(* Schneider Machine Expert - Basic project resolucao, file version 2.7.0.0 *)
(* ProjectInformations: Name=Novo projeto *)

HARDWARE
  Cpu 0: TM221CE24R
  EthernetConfiguration: NetworkName=M221, IpAllocationMode=FixedAddress, IpAddress=0.0.0.0, SubnetMask=0.0.0.0
  SerialLineConfiguration: Baud=Baud19200, Parity=ParityEven, DataBits=DataBits8, StopBits=StopBits1, PhysicalMedium=PhysicalMediumRs485, TransmissionMode=TransmissionModeModbusRtu, SlaveId=1, Addressing=SlaveAddressing
  MastTask: UsePeriodScanMode=false, PeriodScan=100
  FastTask: Period=255
  CpuBehavior: StartingMode=StartAsPreviousState, AutoSaveRamOnEeprom=true, WatchdogPeriod=250

SYMBOLS  (address, symbol, comment, settings)
  %M0       SIG_IN_BOT_G
  %M10      SIG_OUT_CON_A_LIGA
  %M11      SIG_OUT_CON_A_DESL
  %M12      SIG_OUT_MOT_E_LIGA
  %M13      SIG_OUT_MOT_E_DESL
  %TM0      T_CON_A_LIGA  [Preset=5, Base=OneHundredMilliSeconds]
  %TM1        [Preset=5, Base=OneHundredMilliSeconds]
  %I0.0     IN_BOT_G
  %Q0.1     OUT_CON_A
  %Q0.2     OUT_MOT_E

POU Entradas
  (* SectionNumber=1 *)

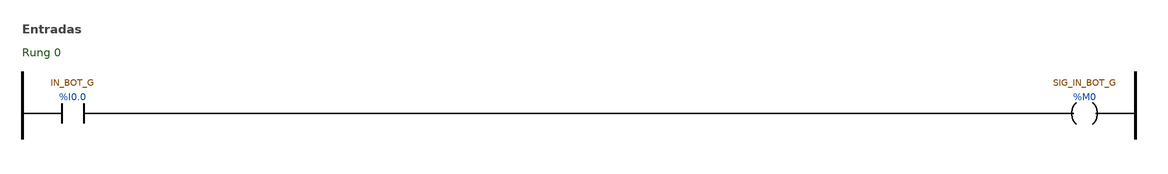

// Rung 0
  LD %I0.0                (* IN_BOT_G *)
  ST %M0                  (* SIG_IN_BOT_G *)
  // as ST:
  //   SIG_IN_BOT_G := IN_BOT_G;

POU Lógicas
  (* SectionNumber=2 *)

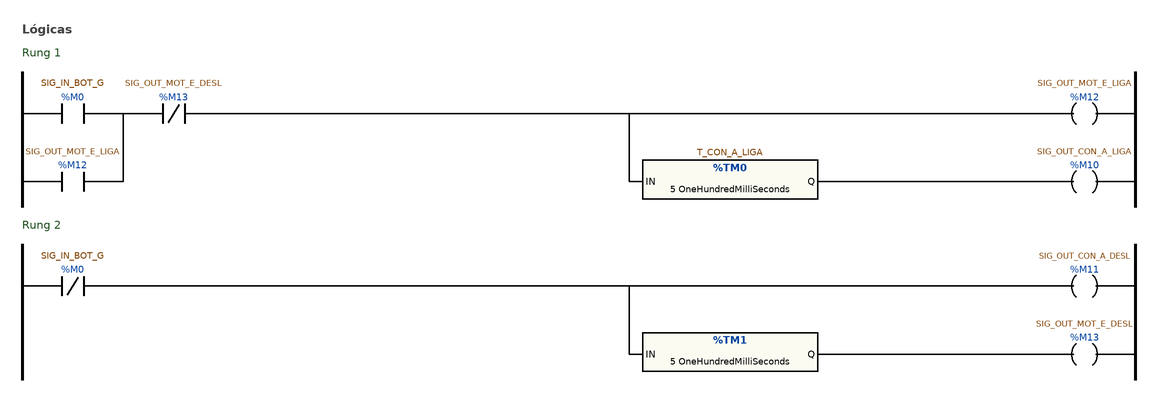

// Rung 1
  LD 1
  MULTIFB
  LD 1
  AND %M0                 (* SIG_IN_BOT_G *)
  OR %M12                 (* SIG_OUT_MOT_E_LIGA *)
  ANDN %M13               (* SIG_OUT_MOT_E_DESL *)
  ST %MW2009:X0
  LD %MW2009:X0
  ST %M12                 (* SIG_OUT_MOT_E_LIGA *)
  BLK %TM0                (* T_CON_A_LIGA *)
  LD %MW2009:X0
  IN
  OUT_BLK
  LD Q
  ST %M10                 (* SIG_OUT_CON_A_LIGA *)
  END_BLK
  MULTIFB
  // as ST:
  //   _t1 := (SIG_IN_BOT_G OR SIG_OUT_MOT_E_LIGA) AND NOT SIG_OUT_MOT_E_DESL;
  //   SIG_OUT_MOT_E_LIGA := _t1;
  //   T_CON_A_LIGA(IN := _t1);
  //   SIG_OUT_CON_A_LIGA := T_CON_A_LIGA.Q;

// Rung 2
  LD 1
  MULTIFB
  LD 1
  ANDN %M0                (* SIG_IN_BOT_G *)
  ST %MW2009:X0
  LD %MW2009:X0
  ST %M11                 (* SIG_OUT_CON_A_DESL *)
  BLK %TM1
  LD %MW2009:X0
  IN
  OUT_BLK
  LD Q
  ST %M13                 (* SIG_OUT_MOT_E_DESL *)
  END_BLK
  MULTIFB
  // as ST:
  //   SIG_OUT_CON_A_DESL := NOT SIG_IN_BOT_G;
  //   %TM1(IN := NOT SIG_IN_BOT_G);
  //   SIG_OUT_MOT_E_DESL := %TM1.Q;

POU Saídas
  (* SectionNumber=3 *)

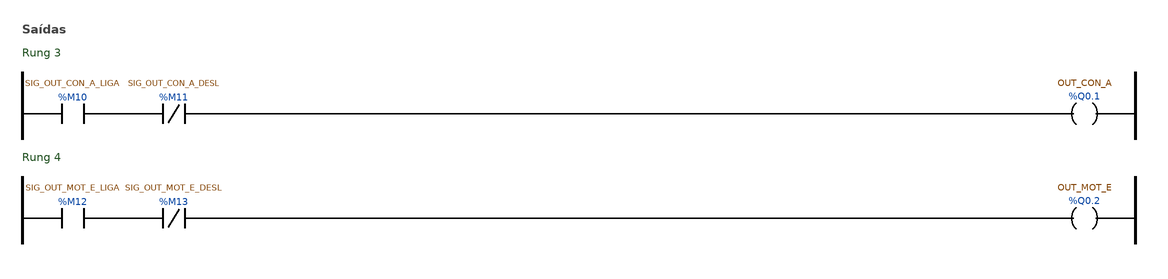

// Rung 3
  LD %M10                 (* SIG_OUT_CON_A_LIGA *)
  ANDN %M11               (* SIG_OUT_CON_A_DESL *)
  ST %Q0.1                (* OUT_CON_A *)
  // as ST:
  //   OUT_CON_A := SIG_OUT_CON_A_LIGA AND NOT SIG_OUT_CON_A_DESL;

// Rung 4
  LD %M12                 (* SIG_OUT_MOT_E_LIGA *)
  ANDN %M13               (* SIG_OUT_MOT_E_DESL *)
  ST %Q0.2                (* OUT_MOT_E *)
  // as ST:
  //   OUT_MOT_E := SIG_OUT_MOT_E_LIGA AND NOT SIG_OUT_MOT_E_DESL;
